Yaskawa INFORM job: test1_tjr0.JBI

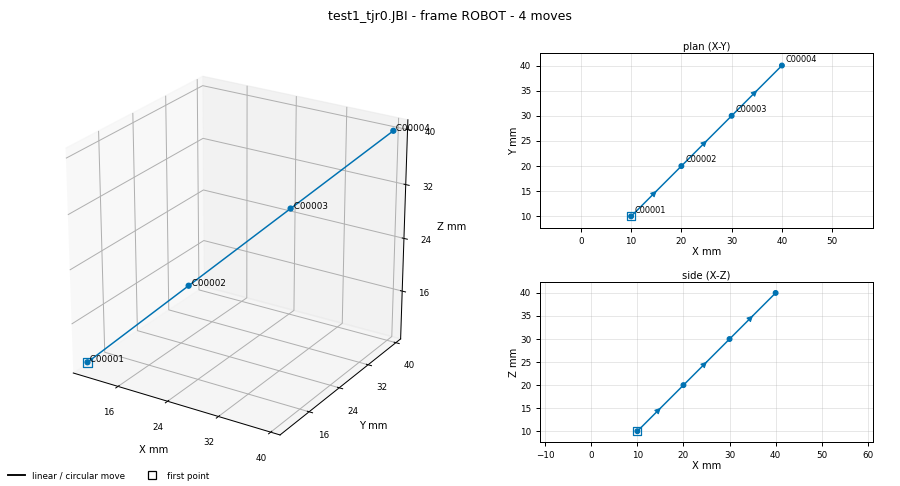
[picture p0: tool path of test1_tjr0.JBI in frame ROBOT, 4 of 5 moves have a stored position in this frame; points joined in program order, loops and branches not executed]
'version: 0
/JOB
//NAME test1
//POS
///NPOS 48,0,0,2,0,0
///TOOL 1
///POSTYPE ROBOT
///RECTAN
///RCONF 1,0,0,0,0,0,0,0,0,0,0,0,0,0,0,0,0,0,0,0,0,0,0,0
C00000=0.000,0.000,0.000,1.0000,0.0000,0.0000
C00001=10.000,10.000,10.000,0.0000,1.0000,0.0000
C00002=20.000,20.000,20.000,0.0000,0.0000,1.0000
C00003=30.000,30.000,30.000,1.0000,0.0000,0.0000
C00004=40.000,40.000,40.000,1.0000,0.0000,0.0000
//INST
///DATE 03/29/2021 17:05
///COMM
///ATTR SC,RW,RJ
///FRAME ROBOT
///GROUP1 RB1
NOP
' first example of file for tool generation
SPEED V=10.2
MOVL C00001
SPEED V=50.0
MOVL C00002
MOVL C00003
TIMER T=10.23
DOUT OG#(12) 1
ARCON
MOVL C00004
ARCOF
MOVL C00005
END
